(* PLC project Tc3_EventLogger.FB_RemoteListenerBase Demo, tc3-libraries-kb TwinCAT 3.1 *)
(* stored: creationDateTime 2026-05-11T01:00:00, modificationDateTime 2026-05-11T01:00:00 *)

PROGRAM P_Demo_FB_RemoteListenerBase
  VAR
    fbFB_RemoteListenerBase : FB_RemoteListenerBase;  (* Tc3_EventLogger.FB_RemoteListenerBase 实例 *)
    arg_ipContext : I_TcListenerContext;  (* VAR_INPUT ipContext *)
    arg_fbEvent : REFERENCE TO FB_TcEvent;  (* VAR_INPUT fbEvent *)
    arg_eReason : TcRemoteConnectionChangeReason;  (* VAR_INPUT eReason *)
    arg_eReason : TcDatabaseChangeReason;  (* VAR_INPUT eReason *)
    arg_hr : HRESULT;  (* VAR_INPUT hr *)
    arg_ipRemoteLogger : I_TcRemoteEventLogger;  (* VAR_INPUT ipRemoteLogger *)
    arg_ipEventFilter : I_TcEventFilterBase;  (* VAR_INPUT ipEventFilter *)
  END_VAR

            // ============================================================
// Tc3_EventLogger.FB_RemoteListenerBase 演示程序（FB 实例）
// ============================================================
// 验证步骤：
//   1. 引用 Tc3_EventLogger（及依赖类型所在库 Tc2_System 等）
//   2. 编译 + 登录
//   3. 按 doc.md 给 arg_* 赋值
//   4. 在线监视 out_* / io_* 输出
// ============================================================

fbFB_RemoteListenerBase(
    ipContext := arg_ipContext,
    fbEvent := arg_fbEvent,
    eReason := arg_eReason,
    eReason := arg_eReason,
    hr := arg_hr,
    ipRemoteLogger := arg_ipRemoteLogger,
    ipEventFilter := arg_ipEventFilter
);

          
END_PROGRAM
